PROGRAM sevenSegProg
VAR
digit1Decoder : SevenSegDecoder;
inputDigit : INT := 0;
END_VAR

digit1Decoder(digit:= inputDigit);

END_PROGRAM

(* stored: Version 1.1.0.1, ProductVersion 3.1.4024.5
   POU sevenSegProg: Id {aa3e8933-31ae-463c-8baf-c27d56345385}, SpecialFunc None *)
